RoboDK station: M301_01 v3.rdk

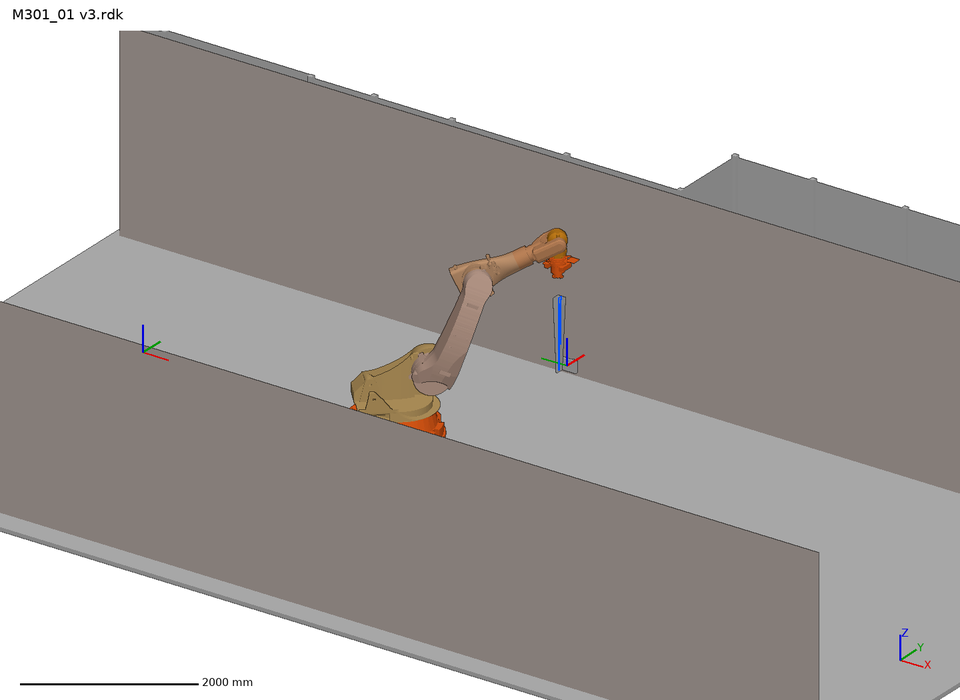
[picture v0: the station drawn from its stored meshes, robots at their saved joint values, targets as dots, program paths as lines]
Station CTTLab. Poses are relative to the parent item; angles as X-Y-Z fixed-axis rotations.
  - object PLANCHER at (0, 0, 0) mm, size 14365 x 8134 x 50 mm, geometry from PLANCHER.STL
  - object BARRIERE_POTEAU at (0, 0, 0) mm, size 13974 x 1274 x 2640 mm, geometry from BARRIERE_POTEAU.STL
  - object BARRIERE_GRILLAGE at (0, 0, 0) mm, size 13811.6 x 1129 x 2475 mm, geometry from BARRIERE_GRILLAGE.STL
  - object BARRIERE_IMMATERIELLE at (0, 0, 0) mm, size 14165 x 6570 x 2640 mm, geometry from BARRIERE_IMMATERIELLE.STL
  - frame World Base at (0, 0, 2.5) mm
    - robot Linear Rail: 1 axes
        modified DH rows (alpha deg, a mm, theta deg, d mm): 0, 0, 0, 0 linear
        base shift (0, 0, 0) mm, rotated rx 0 ry 90 rz 0 deg
        joint limits [0] to [7000]; home [0]; saved at [3500]
      - robot KUKA KR 100 HA: 6 axes
          modified DH rows (alpha deg, a mm, theta deg, d mm): 0, 0, 0, 750; -90, 350, 0, 0; 0, 1250, -90, 0; -90, -45, 0, 1000; 90, 0, 0, 0; -90, 0, 180, 210
          joint limits [-185, -120, -119, -350, -125, -350] to [185, 70, 155, 350, 125, 350]; home [0, -90, 90, 0, 0, 0]; saved at [-41.564, -65.811, 41.041, 0, 114.77, -131.564]
        - tool Tool 1, TCP at (13, 8, 496) mm, size 290.8 x 416.4 x 279.8 mm, geometry from OUTIL.STL
          - object M301_01 at (0, 0, 0) mm, size 101.6 x 101.6 x 914.4 mm, geometry from M301_01.stl
  - frame Camera base at (4846.59, 1350.74, 651.46) mm, rotated rx 0 ry 0 rz 90 deg
    - object Camera at (0, 0, 0) mm, rotated rx 90 ry 0 rz 90 deg, size 220 x 170 x 50 mm, geometry from Camera.stl
    - target Approach target (Cartesian target) at (-112.7, 0, 313.4) mm, rotated rx -180 ry 0 rz -90 deg; joints [-43.056, -66.41, 76.951, 0, 79.459, 136.944, 3500] of KUKA KR 100 HA
    - target Target 0 (Cartesian target) at (-112.7, 0, 881.94) mm, rotated rx -180 ry 0 rz -90 deg; joints [-43.056, -64.348, 40.687, 0, 113.661, 136.944, 3500] of KUKA KR 100 HA
    - target Target 1 (Cartesian target) at (-124.95, 0, 850.56) mm, rotated rx -180 ry 0 rz -90 deg; joints [-42.537, -65.949, 45.083, -0.648, 110.311, 137.463, 3500] of KUKA KR 100 HA
    - target Target 2 (Cartesian target) at (-139.47, 0, 817.45) mm, rotated rx -177.14 ry 0 rz -90 deg; joints [-41.911, -67.558, 49.528, -1.405, 106.807, 137.413, 3500] of KUKA KR 100 HA
    - target Target 3 (Cartesian target) at (-154.54, 0, 817.31) mm, rotated rx -177.14 ry 0 rz -90 deg; joints [-41.235, -68.595, 51.082, -2.235, 105.614, 138.127, 3500] of KUKA KR 100 HA
    - target Target 4 (Cartesian target) at (-154.54, 0, 785.81) mm, rotated rx -177.14 ry 0 rz -90 deg; joints [-41.235, -69.02, 53.562, -2.214, 103.561, 138.21, 3500] of KUKA KR 100 HA
    - target Target 5 (Cartesian target) at (-154.54, 0, 785.81) mm, rotated rx -177.14 ry 0 rz -90 deg; joints [-41.235, -69.02, 53.562, -2.214, 103.561, 138.21, 3500] of KUKA KR 100 HA
    - target Target 6 (Cartesian target) at (-154.54, 0, 754.31) mm, rotated rx -177.14 ry 0 rz -90 deg; joints [-41.235, -69.373, 55.917, -2.197, 101.559, 138.289, 3500] of KUKA KR 100 HA
    - target Target 7 (Cartesian target) at (-154.54, 0, 754.31) mm, rotated rx -177.14 ry 0 rz -90 deg; joints [-41.235, -69.373, 55.917, -2.197, 101.559, 138.289, 3500] of KUKA KR 100 HA
    - target Target 8 (Cartesian target) at (-154.54, 0, 722.81) mm, rotated rx -177.14 ry 0 rz -90 deg; joints [-41.235, -69.661, 58.163, -2.183, 99.603, 138.365, 3500] of KUKA KR 100 HA
    - target Target 9 (Cartesian target) at (-154.54, 0, 722.81) mm, rotated rx -177.14 ry 0 rz -90 deg; joints [-41.235, -69.661, 58.163, -2.183, 99.603, 138.365, 3500] of KUKA KR 100 HA
    - target Target 10 (Cartesian target) at (-154.54, 0, 691.3) mm, rotated rx -177.14 ry 0 rz -90 deg; joints [-41.235, -69.887, 60.31, -2.172, 97.685, 138.439, 3500] of KUKA KR 100 HA
    - target Target 11 (Cartesian target) at (-154.54, 0, 691.3) mm, rotated rx -177.14 ry 0 rz -90 deg; joints [-41.235, -69.887, 60.31, -2.172, 97.685, 138.439, 3500] of KUKA KR 100 HA
    - target Target 12 (Cartesian target) at (-154.54, 0, 659.8) mm, rotated rx -177.14 ry 0 rz -90 deg; joints [-41.235, -70.057, 62.366, -2.163, 95.8, 138.51, 3500] of KUKA KR 100 HA
    - target Target 13 (Cartesian target) at (-154.54, 0, 659.8) mm, rotated rx -177.14 ry 0 rz -90 deg; joints [-41.235, -70.057, 62.366, -2.163, 95.8, 138.51, 3500] of KUKA KR 100 HA
    - target Target 14 (Cartesian target) at (-154.54, 0, 628.3) mm, rotated rx -177.14 ry 0 rz -90 deg; joints [-41.235, -70.173, 64.338, -2.157, 93.944, 138.581, 3500] of KUKA KR 100 HA
    - target Target 15 (Cartesian target) at (-154.54, 0, 628.3) mm, rotated rx -177.14 ry 0 rz -90 deg; joints [-41.235, -70.173, 64.338, -2.157, 93.944, 138.581, 3500] of KUKA KR 100 HA
    - target Target 16 (Cartesian target) at (-154.54, 0, 596.8) mm, rotated rx -177.14 ry 0 rz -90 deg; joints [-41.235, -70.236, 66.234, -2.154, 92.114, 138.65, 3500] of KUKA KR 100 HA
    - target Target 17 (Cartesian target) at (-154.54, 0, 596.8) mm, rotated rx -177.14 ry 0 rz -90 deg; joints [-41.235, -70.236, 66.234, -2.154, 92.114, 138.65, 3500] of KUKA KR 100 HA
    - target Target 18 (Cartesian target) at (-154.54, 0, 565.3) mm, rotated rx -177.14 ry 0 rz -90 deg; joints [-41.235, -70.25, 68.057, -2.152, 90.306, 138.718, 3500] of KUKA KR 100 HA
    - target Target 19 (Cartesian target) at (-154.54, 0, 565.3) mm, rotated rx -177.14 ry 0 rz -90 deg; joints [-41.235, -70.25, 68.057, -2.152, 90.306, 138.718, 3500] of KUKA KR 100 HA
    - target Target 20 (Cartesian target) at (-154.54, 0, 533.8) mm, rotated rx -177.14 ry 0 rz -90 deg; joints [-41.235, -70.216, 69.812, -2.153, 88.518, 138.785, 3500] of KUKA KR 100 HA
    - target Target 21 (Cartesian target) at (-154.54, 0, 533.8) mm, rotated rx -177.14 ry 0 rz -90 deg; joints [-41.235, -70.216, 69.812, -2.153, 88.518, 138.785, 3500] of KUKA KR 100 HA
    - target Target 22 (Cartesian target) at (-154.54, 0, 502.3) mm, rotated rx -177.14 ry 0 rz -90 deg; joints [-41.235, -70.136, 71.503, -2.156, 86.747, 138.851, 3500] of KUKA KR 100 HA
    - target Target 23 (Cartesian target) at (-154.54, 0, 502.3) mm, rotated rx -177.14 ry 0 rz -90 deg; joints [-41.235, -70.136, 71.503, -2.156, 86.747, 138.851, 3500] of KUKA KR 100 HA
    - target Target 24 (Cartesian target) at (-154.54, 0, 470.79) mm, rotated rx -177.14 ry 0 rz -90 deg; joints [-41.235, -70.01, 73.133, -2.16, 84.993, 138.918, 3500] of KUKA KR 100 HA
    - target Target 25 (Cartesian target) at (-154.54, 0, 470.79) mm, rotated rx -177.14 ry 0 rz -90 deg; joints [-41.235, -70.01, 73.133, -2.16, 84.993, 138.918, 3500] of KUKA KR 100 HA
    - target Target 26 (Cartesian target) at (-154.54, 0, 439.29) mm, rotated rx -177.14 ry 0 rz -90 deg; joints [-41.235, -69.84, 74.705, -2.167, 83.252, 138.984, 3500] of KUKA KR 100 HA
    - target Target 27 (Cartesian target) at (-154.54, 0, 439.29) mm, rotated rx -177.14 ry 0 rz -90 deg; joints [-41.235, -69.84, 74.705, -2.167, 83.252, 138.984, 3500] of KUKA KR 100 HA
    - target Target 28 (Cartesian target) at (-154.54, 0, 407.79) mm, rotated rx -177.14 ry 0 rz -90 deg; joints [-41.235, -69.627, 76.221, -2.176, 81.524, 139.05, 3500] of KUKA KR 100 HA
    - target Target 29 (Cartesian target) at (-154.54, 0, 407.79) mm, rotated rx -177.14 ry 0 rz -90 deg; joints [-41.235, -69.627, 76.221, -2.176, 81.524, 139.05, 3500] of KUKA KR 100 HA
    - target Target 30 (Cartesian target) at (-154.54, 0, 376.29) mm, rotated rx -177.14 ry 0 rz -90 deg; joints [-41.235, -69.371, 77.683, -2.187, 79.808, 139.116, 3500] of KUKA KR 100 HA
    - target Target 31 (Cartesian target) at (-154.54, 0, 376.29) mm, rotated rx -177.14 ry 0 rz -90 deg; joints [-41.235, -69.371, 77.683, -2.187, 79.808, 139.116, 3500] of KUKA KR 100 HA
    - target Target 32 (Cartesian target) at (-154.54, 0, 344.79) mm, rotated rx -177.14 ry 0 rz -90 deg; joints [-41.235, -69.074, 79.092, -2.199, 78.102, 139.183, 3500] of KUKA KR 100 HA
    - target Target 33 (Cartesian target) at (-154.54, 0, 344.79) mm, rotated rx -177.14 ry 0 rz -90 deg; joints [-41.235, -69.074, 79.092, -2.199, 78.102, 139.183, 3500] of KUKA KR 100 HA
    - target Target 34 (Cartesian target) at (-154.54, 0, 313.29) mm, rotated rx -177.14 ry 0 rz -90 deg; joints [-41.235, -68.735, 80.451, -2.214, 76.406, 139.25, 3500] of KUKA KR 100 HA
    - target Target 35 (Cartesian target) at (-154.54, 0, 313.29) mm, rotated rx -177.14 ry 0 rz -90 deg; joints [-41.235, -68.735, 80.451, -2.214, 76.406, 139.25, 3500] of KUKA KR 100 HA
    - target Target 36 (Cartesian target) at (-154.54, 0, 281.79) mm, rotated rx -177.14 ry 0 rz -90 deg; joints [-41.235, -68.356, 81.76, -2.231, 74.719, 139.317, 3500] of KUKA KR 100 HA
    - target Target 37 (Cartesian target) at (-154.54, 0, 281.79) mm, rotated rx -177.14 ry 0 rz -90 deg; joints [-41.235, -68.356, 81.76, -2.231, 74.719, 139.317, 3500] of KUKA KR 100 HA
    - target Target 38 (Cartesian target) at (-154.54, 0, 250.29) mm, rotated rx -177.14 ry 0 rz -90 deg; joints [-41.235, -67.936, 83.021, -2.25, 73.04, 139.386, 3500] of KUKA KR 100 HA
    - target Target 39 (Cartesian target) at (-154.54, 0, 218.78) mm, rotated rx -177.14 ry 0 rz -90 deg; joints [-41.235, -67.477, 84.234, -2.271, 71.37, 139.455, 3500] of KUKA KR 100 HA
    - target Target 40 (Cartesian target) at (-154.54, 0, 218.78) mm, rotated rx -177.14 ry 0 rz -90 deg; joints [-41.235, -67.477, 84.234, -2.271, 71.37, 139.455, 3500] of KUKA KR 100 HA
    - target Target 41 (Cartesian target) at (-154.54, 0, 187.28) mm, rotated rx -177.14 ry 0 rz -90 deg; joints [-41.235, -66.979, 85.4, -2.295, 69.707, 139.525, 3500] of KUKA KR 100 HA
    - target Target 42 (Cartesian target) at (-154.54, 0, 187.28) mm, rotated rx -177.14 ry 0 rz -90 deg; joints [-41.235, -66.979, 85.4, -2.295, 69.707, 139.525, 3500] of KUKA KR 100 HA
    - target Target 43 (Cartesian target) at (-154.54, 0, 155.78) mm, rotated rx -177.14 ry 0 rz -90 deg; joints [-41.235, -66.442, 86.519, -2.32, 68.051, 139.597, 3500] of KUKA KR 100 HA
    - target Target 44 (Cartesian target) at (-154.54, 0, 155.78) mm, rotated rx -177.14 ry 0 rz -90 deg; joints [-41.235, -66.442, 86.519, -2.32, 68.051, 139.597, 3500] of KUKA KR 100 HA
    - target Target 45 (Cartesian target) at (-154.54, 0, 124.28) mm, rotated rx -177.14 ry 0 rz -90 deg; joints [-41.235, -65.867, 87.593, -2.349, 66.403, 139.67, 3500] of KUKA KR 100 HA
    - target Target 46 (Cartesian target) at (-154.54, 0, 124.28) mm, rotated rx -177.14 ry 0 rz -90 deg; joints [-41.235, -65.867, 87.593, -2.349, 66.403, 139.67, 3500] of KUKA KR 100 HA
    - target Target 47 (Cartesian target) at (-154.54, 0, 92.78) mm, rotated rx -177.14 ry 0 rz -90 deg; joints [-41.235, -65.254, 88.622, -2.379, 64.763, 139.744, 3500] of KUKA KR 100 HA
    - target Target 48 (Cartesian target) at (-152.66, 0, 92.8) mm, rotated rx -177.14 ry 0 rz -90 deg; joints [-41.626, -64.816, 87.917, -1.397, 65.788, 139.307, 3500] of KUKA KR 100 HA
    - target Target 49 (Cartesian target) at (-151.82, 0, 63.93) mm, rotated rx -180 ry 0 rz -90 deg; joints [-41.878, -63.949, 88.344, -0.751, 64.989, 138.122, 3500] of KUKA KR 100 HA
    - target Target 50 (Cartesian target) at (-150.8, 0, 32.46) mm, rotated rx -180 ry 0 rz -90 deg; joints [-42.17, -62.942, 88.744, 0, 64.199, 137.83, 3500] of KUKA KR 100 HA
    - target Target 51 (Cartesian target) at (-150.8, 0, 1) mm, rotated rx -180 ry 0 rz -90 deg; joints [-42.17, -62.239, 89.64, 0, 62.599, 137.83, 3500] of KUKA KR 100 HA
    - target Target 52 (Cartesian target) at (-150.8, 0, 1) mm, rotated rx -180 ry 0 rz 180 deg; joints [-41.842, -61.484, 88.373, 0, 63.111, 48.158, 3500] of KUKA KR 100 HA
    - target Target 53 (Cartesian target) at (-150.8, 0, 32.46) mm, rotated rx -180 ry 0 rz 180 deg; joints [-41.842, -62.176, 87.478, 0, 64.699, 48.158, 3500] of KUKA KR 100 HA
    - target Target 54 (Cartesian target) at (-150.8, 0, 63.92) mm, rotated rx -180 ry 0 rz 180 deg; joints [-41.842, -62.833, 86.537, 0, 66.296, 48.158, 3500] of KUKA KR 100 HA
    - target Target 55 (Cartesian target) at (-150.8, 0, 95.39) mm, rotated rx -180 ry 0 rz 180 deg; joints [-41.842, -63.453, 85.55, 0, 67.903, 48.158, 3500] of KUKA KR 100 HA
    - target Target 56 (Cartesian target) at (-150.8, 0, 126.85) mm, rotated rx -180 ry 0 rz 180 deg; joints [-41.842, -64.037, 84.517, 0, 69.52, 48.158, 3500] of KUKA KR 100 HA
    - target Target 57 (Cartesian target) at (-150.8, 0, 158.31) mm, rotated rx -180 ry 0 rz 180 deg; joints [-41.842, -64.584, 83.438, 0, 71.146, 48.158, 3500] of KUKA KR 100 HA
    - target Target 58 (Cartesian target) at (-150.8, 0, 189.77) mm, rotated rx -180 ry 0 rz 180 deg; joints [-41.842, -65.094, 82.313, 0, 72.781, 48.158, 3500] of KUKA KR 100 HA
    - target Target 59 (Cartesian target) at (-150.8, 0, 221.23) mm, rotated rx -180 ry 0 rz 180 deg; joints [-41.842, -65.565, 81.139, 0, 74.426, 48.158, 3500] of KUKA KR 100 HA
    - target Target 60 (Cartesian target) at (-150.8, 0, 252.7) mm, rotated rx -180 ry 0 rz 180 deg; joints [-41.842, -65.997, 79.917, 0, 76.08, 48.158, 3500] of KUKA KR 100 HA
    - target Target 61 (Cartesian target) at (-150.8, 0, 284.16) mm, rotated rx -180 ry 0 rz 180 deg; joints [-41.842, -66.391, 78.646, 0, 77.744, 48.158, 3500] of KUKA KR 100 HA
    - target Target 62 (Cartesian target) at (-150.8, 0, 315.62) mm, rotated rx -180 ry 0 rz 180 deg; joints [-41.842, -66.744, 77.325, 0, 79.419, 48.158, 3500] of KUKA KR 100 HA
    - target Target 63 (Cartesian target) at (-150.8, 0, 347.08) mm, rotated rx -180 ry 0 rz 180 deg; joints [-41.842, -67.057, 75.952, 0, 81.106, 48.158, 3500] of KUKA KR 100 HA
    - target Target 64 (Cartesian target) at (-150.8, 0, 378.54) mm, rotated rx -180 ry 0 rz 180 deg; joints [-41.842, -67.329, 74.525, 0, 82.804, 48.158, 3500] of KUKA KR 100 HA
    - target Target 65 (Cartesian target) at (-150.8, 0, 410.01) mm, rotated rx -180 ry 0 rz 180 deg; joints [-41.842, -67.559, 73.044, 0, 84.515, 48.158, 3500] of KUKA KR 100 HA
    - target Target 66 (Cartesian target) at (-150.8, 0, 441.47) mm, rotated rx -180 ry 0 rz 180 deg; joints [-41.842, -67.746, 71.505, 0, 86.241, 48.158, 3500] of KUKA KR 100 HA
    - target Target 67 (Cartesian target) at (-150.8, 0, 472.93) mm, rotated rx -180 ry 0 rz 180 deg; joints [-41.842, -67.89, 69.908, 0, 87.982, 48.158, 3500] of KUKA KR 100 HA
    - target Target 68 (Cartesian target) at (-150.8, 0, 504.39) mm, rotated rx -180 ry 0 rz 180 deg; joints [-41.842, -67.988, 68.248, 0, 89.741, 48.158, 3500] of KUKA KR 100 HA
    - target Target 69 (Cartesian target) at (-150.8, 0, 535.86) mm, rotated rx -180 ry 0 rz 180 deg; joints [-41.842, -68.04, 66.522, 0, 91.518, 48.158, 3500] of KUKA KR 100 HA
    - target Target 70 (Cartesian target) at (-150.8, 0, 567.32) mm, rotated rx -180 ry 0 rz 180 deg; joints [-41.842, -68.045, 64.728, 0, 93.317, 48.158, 3500] of KUKA KR 100 HA
    - target Target 71 (Cartesian target) at (-150.8, 0, 598.78) mm, rotated rx -180 ry 0 rz 180 deg; joints [-41.842, -67.999, 62.86, 0, 95.14, 48.158, 3500] of KUKA KR 100 HA
    - target Target 72 (Cartesian target) at (-150.8, 0, 630.24) mm, rotated rx -180 ry 0 rz 180 deg; joints [-41.842, -67.902, 60.912, 0, 96.99, 48.158, 3500] of KUKA KR 100 HA
    - target Target 73 (Cartesian target) at (-150.8, 0, 661.7) mm, rotated rx -180 ry 0 rz 180 deg; joints [-41.842, -67.75, 58.88, 0, 98.87, 48.158, 3500] of KUKA KR 100 HA
    - target Target 74 (Cartesian target) at (-150.8, 0, 693.17) mm, rotated rx -180 ry 0 rz 180 deg; joints [-41.842, -67.541, 56.755, 0, 100.786, 48.158, 3500] of KUKA KR 100 HA
    - target Target 75 (Cartesian target) at (-150.8, 0, 724.63) mm, rotated rx -180 ry 0 rz 180 deg; joints [-41.842, -67.27, 54.528, 0, 102.742, 48.158, 3500] of KUKA KR 100 HA
    - target Target 76 (Cartesian target) at (-150.8, 0, 756.09) mm, rotated rx -180 ry 0 rz 180 deg; joints [-41.842, -66.933, 52.188, 0, 104.745, 48.158, 3500] of KUKA KR 100 HA
    - target Target 77 (Cartesian target) at (-150.8, 0, 787.55) mm, rotated rx -180 ry 0 rz 180 deg; joints [-41.842, -66.524, 49.722, 0, 106.802, 48.158, 3500] of KUKA KR 100 HA
    - target Target 78 (Cartesian target) at (-150.8, 0, 819.01) mm, rotated rx -180 ry 0 rz 180 deg; joints [-41.842, -66.034, 47.111, 0, 108.924, 48.158, 3500] of KUKA KR 100 HA
    - target Target 79 (Cartesian target) at (-150.8, 0, 850.48) mm, rotated rx -180 ry 0 rz 180 deg; joints [-41.842, -65.455, 44.332, 0, 111.123, 48.158, 3500] of KUKA KR 100 HA
    - target Target 80 (Cartesian target) at (-150.8, 0, 881.94) mm, rotated rx -180 ry 0 rz 180 deg; joints [-41.842, -64.773, 41.356, 0, 113.417, 48.158, 3500] of KUKA KR 100 HA
    - target Target 81 (Cartesian target) at (-150.8, 0, 913.4) mm, rotated rx -180 ry 0 rz 180 deg; joints [-41.842, -63.969, 38.141, 0, 115.828, 48.158, 3500] of KUKA KR 100 HA
    - target Target 82 (Cartesian target) at (-112.7, 0, 913.4) mm, rotated rx -180 ry 0 rz 90 deg; joints [-42.136, -62.977, 36.545, 0, 116.432, -42.136, 3500] of KUKA KR 100 HA
    - target Target 83 (Cartesian target) at (-112.7, 0, 881.94) mm, rotated rx -180 ry 0 rz 90 deg; joints [-42.136, -63.826, 39.86, 0, 113.966, -42.136, 3500] of KUKA KR 100 HA
    - target Target 84 (Cartesian target) at (-124.95, 0, 850.56) mm, rotated rx -180 ry 0 rz 90 deg; joints [-41.612, -65.441, 44.3, -0.659, 110.596, -41.612, 3500] of KUKA KR 100 HA
    - target Target 85 (Cartesian target) at (-139.47, 0, 817.45) mm, rotated rx 177.14 ry 0 rz 90 deg; joints [-40.979, -67.07, 48.843, -1.427, 107.026, -41.674, 3500] of KUKA KR 100 HA
    - target Target 86 (Cartesian target) at (-154.54, 0, 817.31) mm, rotated rx 177.14 ry 0 rz 90 deg; joints [-40.298, -68.096, 50.392, -2.269, 105.84, -40.953, 3500] of KUKA KR 100 HA
    - target Target 87 (Cartesian target) at (-154.54, 0, 785.81) mm, rotated rx 177.14 ry 0 rz 90 deg; joints [-40.298, -68.53, 52.891, -2.247, 103.776, -40.869, 3500] of KUKA KR 100 HA
    - target Target 88 (Cartesian target) at (-154.54, 0, 785.81) mm, rotated rx 177.14 ry 0 rz 90 deg; joints [-40.298, -68.53, 52.891, -2.247, 103.776, -40.869, 3500] of KUKA KR 100 HA
    - target Target 89 (Cartesian target) at (-154.54, 0, 754.31) mm, rotated rx 177.14 ry 0 rz 90 deg; joints [-40.298, -68.891, 55.263, -2.23, 101.766, -40.788, 3500] of KUKA KR 100 HA
    - target Target 90 (Cartesian target) at (-154.54, 0, 754.31) mm, rotated rx 177.14 ry 0 rz 90 deg; joints [-40.298, -68.891, 55.263, -2.23, 101.766, -40.788, 3500] of KUKA KR 100 HA
    - target Target 91 (Cartesian target) at (-154.54, 0, 722.81) mm, rotated rx 177.14 ry 0 rz 90 deg; joints [-40.298, -69.185, 57.523, -2.215, 99.803, -40.711, 3500] of KUKA KR 100 HA
    - target Target 92 (Cartesian target) at (-154.54, 0, 722.81) mm, rotated rx 177.14 ry 0 rz 90 deg; joints [-40.298, -69.185, 57.523, -2.215, 99.803, -40.711, 3500] of KUKA KR 100 HA
    - target Target 93 (Cartesian target) at (-154.54, 0, 691.3) mm, rotated rx 177.14 ry 0 rz 90 deg; joints [-40.298, -69.418, 59.681, -2.204, 97.879, -40.636, 3500] of KUKA KR 100 HA
    - target Target 94 (Cartesian target) at (-154.54, 0, 691.3) mm, rotated rx 177.14 ry 0 rz 90 deg; joints [-40.298, -69.418, 59.681, -2.204, 97.879, -40.636, 3500] of KUKA KR 100 HA
    - target Target 95 (Cartesian target) at (-154.54, 0, 659.8) mm, rotated rx 177.14 ry 0 rz 90 deg; joints [-40.298, -69.593, 61.747, -2.195, 95.99, -40.563, 3500] of KUKA KR 100 HA
    - target Target 96 (Cartesian target) at (-154.54, 0, 659.8) mm, rotated rx 177.14 ry 0 rz 90 deg; joints [-40.298, -69.593, 61.747, -2.195, 95.99, -40.563, 3500] of KUKA KR 100 HA
    - target Target 97 (Cartesian target) at (-154.54, 0, 628.3) mm, rotated rx 177.14 ry 0 rz 90 deg; joints [-40.298, -69.713, 63.728, -2.188, 94.13, -40.491, 3500] of KUKA KR 100 HA
    - target Target 98 (Cartesian target) at (-154.54, 0, 628.3) mm, rotated rx 177.14 ry 0 rz 90 deg; joints [-40.298, -69.713, 63.728, -2.188, 94.13, -40.491, 3500] of KUKA KR 100 HA
    - target Target 99 (Cartesian target) at (-154.54, 0, 596.8) mm, rotated rx 177.14 ry 0 rz 90 deg; joints [-40.298, -69.781, 65.63, -2.184, 92.297, -40.421, 3500] of KUKA KR 100 HA
    - target Target 100 (Cartesian target) at (-154.54, 0, 596.8) mm, rotated rx 177.14 ry 0 rz 90 deg; joints [-40.298, -69.781, 65.63, -2.184, 92.297, -40.421, 3500] of KUKA KR 100 HA
    - target Target 101 (Cartesian target) at (-154.54, 0, 565.3) mm, rotated rx 177.14 ry 0 rz 90 deg; joints [-40.298, -69.8, 67.459, -2.183, 90.488, -40.352, 3500] of KUKA KR 100 HA
    - target Target 102 (Cartesian target) at (-154.54, 0, 565.3) mm, rotated rx 177.14 ry 0 rz 90 deg; joints [-40.298, -69.8, 67.459, -2.183, 90.488, -40.352, 3500] of KUKA KR 100 HA
    - target Target 103 (Cartesian target) at (-154.54, 0, 533.8) mm, rotated rx 177.14 ry 0 rz 90 deg; joints [-40.298, -69.769, 69.22, -2.183, 88.698, -40.284, 3500] of KUKA KR 100 HA
    - target Target 104 (Cartesian target) at (-154.54, 0, 533.8) mm, rotated rx 177.14 ry 0 rz 90 deg; joints [-40.298, -69.769, 69.22, -2.183, 88.698, -40.284, 3500] of KUKA KR 100 HA
    - target Target 105 (Cartesian target) at (-154.54, 0, 502.3) mm, rotated rx 177.14 ry 0 rz 90 deg; joints [-40.298, -69.692, 70.915, -2.186, 86.928, -40.216, 3500] of KUKA KR 100 HA
    - target Target 106 (Cartesian target) at (-154.54, 0, 502.3) mm, rotated rx 177.14 ry 0 rz 90 deg; joints [-40.298, -69.692, 70.915, -2.186, 86.928, -40.216, 3500] of KUKA KR 100 HA
    - target Target 107 (Cartesian target) at (-154.54, 0, 470.79) mm, rotated rx 177.14 ry 0 rz 90 deg; joints [-40.298, -69.57, 72.548, -2.191, 85.173, -40.149, 3500] of KUKA KR 100 HA
    - target Target 108 (Cartesian target) at (-154.54, 0, 470.79) mm, rotated rx 177.14 ry 0 rz 90 deg; joints [-40.298, -69.57, 72.548, -2.191, 85.173, -40.149, 3500] of KUKA KR 100 HA
    - target Target 109 (Cartesian target) at (-154.54, 0, 439.29) mm, rotated rx 177.14 ry 0 rz 90 deg; joints [-40.298, -69.404, 74.123, -2.197, 83.433, -40.082, 3500] of KUKA KR 100 HA
    - target Target 110 (Cartesian target) at (-154.54, 0, 439.29) mm, rotated rx 177.14 ry 0 rz 90 deg; joints [-40.298, -69.404, 74.123, -2.197, 83.433, -40.082, 3500] of KUKA KR 100 HA
    - target Target 111 (Cartesian target) at (-154.54, 0, 407.79) mm, rotated rx 177.14 ry 0 rz 90 deg; joints [-40.298, -69.194, 75.641, -2.206, 81.706, -40.015, 3500] of KUKA KR 100 HA
    - target Target 112 (Cartesian target) at (-154.54, 0, 407.79) mm, rotated rx 177.14 ry 0 rz 90 deg; joints [-40.298, -69.194, 75.641, -2.206, 81.706, -40.015, 3500] of KUKA KR 100 HA
    - target Target 113 (Cartesian target) at (-154.54, 0, 376.29) mm, rotated rx 177.14 ry 0 rz 90 deg; joints [-40.298, -68.941, 77.104, -2.216, 79.992, -39.948, 3500] of KUKA KR 100 HA
    - target Target 114 (Cartesian target) at (-154.54, 0, 376.29) mm, rotated rx 177.14 ry 0 rz 90 deg; joints [-40.298, -68.941, 77.104, -2.216, 79.992, -39.948, 3500] of KUKA KR 100 HA
    - target Target 115 (Cartesian target) at (-154.54, 0, 344.79) mm, rotated rx 177.14 ry 0 rz 90 deg; joints [-40.298, -68.647, 78.515, -2.229, 78.288, -39.881, 3500] of KUKA KR 100 HA
    - target Target 116 (Cartesian target) at (-154.54, 0, 344.79) mm, rotated rx 177.14 ry 0 rz 90 deg; joints [-40.298, -68.647, 78.515, -2.229, 78.288, -39.881, 3500] of KUKA KR 100 HA
    - target Target 117 (Cartesian target) at (-154.54, 0, 313.29) mm, rotated rx 177.14 ry 0 rz 90 deg; joints [-40.298, -68.311, 79.875, -2.244, 76.594, -39.813, 3500] of KUKA KR 100 HA
    - target Target 118 (Cartesian target) at (-154.54, 0, 313.29) mm, rotated rx 177.14 ry 0 rz 90 deg; joints [-40.298, -68.311, 79.875, -2.244, 76.594, -39.813, 3500] of KUKA KR 100 HA
    - target Target 119 (Cartesian target) at (-154.54, 0, 281.79) mm, rotated rx 177.14 ry 0 rz 90 deg; joints [-40.298, -67.935, 81.184, -2.261, 74.91, -39.745, 3500] of KUKA KR 100 HA
    - target Target 120 (Cartesian target) at (-154.54, 0, 281.79) mm, rotated rx 177.14 ry 0 rz 90 deg; joints [-40.298, -67.935, 81.184, -2.261, 74.91, -39.745, 3500] of KUKA KR 100 HA
    - target Target 121 (Cartesian target) at (-154.54, 0, 250.29) mm, rotated rx 177.14 ry 0 rz 90 deg; joints [-40.298, -67.519, 82.445, -2.28, 73.235, -39.676, 3500] of KUKA KR 100 HA
    - target Target 122 (Cartesian target) at (-154.54, 0, 218.78) mm, rotated rx 177.14 ry 0 rz 90 deg; joints [-40.298, -67.064, 83.657, -2.301, 71.568, -39.606, 3500] of KUKA KR 100 HA
    - target Target 123 (Cartesian target) at (-154.54, 0, 218.78) mm, rotated rx 177.14 ry 0 rz 90 deg; joints [-40.298, -67.064, 83.657, -2.301, 71.568, -39.606, 3500] of KUKA KR 100 HA
    - target Target 124 (Cartesian target) at (-154.54, 0, 187.28) mm, rotated rx 177.14 ry 0 rz 90 deg; joints [-40.298, -66.569, 84.823, -2.324, 69.909, -39.535, 3500] of KUKA KR 100 HA
    - target Target 125 (Cartesian target) at (-154.54, 0, 187.28) mm, rotated rx 177.14 ry 0 rz 90 deg; joints [-40.298, -66.569, 84.823, -2.324, 69.909, -39.535, 3500] of KUKA KR 100 HA
    - target Target 126 (Cartesian target) at (-154.54, 0, 155.78) mm, rotated rx 177.14 ry 0 rz 90 deg; joints [-40.298, -66.036, 85.942, -2.35, 68.259, -39.463, 3500] of KUKA KR 100 HA
    - target Target 127 (Cartesian target) at (-154.54, 0, 155.78) mm, rotated rx 177.14 ry 0 rz 90 deg; joints [-40.298, -66.036, 85.942, -2.35, 68.259, -39.463, 3500] of KUKA KR 100 HA
    - target Target 128 (Cartesian target) at (-154.54, 0, 124.28) mm, rotated rx 177.14 ry 0 rz 90 deg; joints [-40.298, -65.465, 87.015, -2.378, 66.616, -39.389, 3500] of KUKA KR 100 HA
    - target Target 129 (Cartesian target) at (-154.54, 0, 124.28) mm, rotated rx 177.14 ry 0 rz 90 deg; joints [-40.298, -65.465, 87.015, -2.378, 66.616, -39.389, 3500] of KUKA KR 100 HA
    - target Target 130 (Cartesian target) at (-154.54, 0, 92.78) mm, rotated rx 177.14 ry 0 rz 90 deg; joints [-40.298, -64.856, 88.042, -2.409, 64.981, -39.314, 3500] of KUKA KR 100 HA
    - target Target 131 (Cartesian target) at (-152.66, 0, 92.8) mm, rotated rx 177.14 ry 0 rz 90 deg; joints [-40.692, -64.426, 87.347, -1.415, 65.989, -39.754, 3500] of KUKA KR 100 HA
    - target Target 132 (Cartesian target) at (-151.82, 0, 63.93) mm, rotated rx -180 ry 0 rz 90 deg; joints [-40.946, -63.584, 87.754, -0.761, 65.226, -40.946, 3500] of KUKA KR 100 HA
    - target Target 133 (Cartesian target) at (-150.8, 0, 32.46) mm, rotated rx -180 ry 0 rz 90 deg; joints [-41.241, -62.589, 88.16, 0, 64.429, -41.241, 3500] of KUKA KR 100 HA
    - target Target 134 (Cartesian target) at (-150.8, 0, 1) mm, rotated rx -180 ry 0 rz 90 deg; joints [-41.241, -61.89, 89.056, 0, 62.835, -41.241, 3500] of KUKA KR 100 HA
    - target Target 135 (Cartesian target) at (-150.8, 0, 1) mm, rotated rx -180 ry 0 rz 0 deg; joints [-41.564, -62.648, 90.321, 0, 62.327, -131.564, 3500] of KUKA KR 100 HA
    - target Target 136 (Cartesian target) at (-150.8, 0, 32.46) mm, rotated rx -180 ry 0 rz 0 deg; joints [-41.564, -63.357, 89.424, 0, 63.933, -131.564, 3500] of KUKA KR 100 HA
    - target Target 137 (Cartesian target) at (-150.8, 0, 63.92) mm, rotated rx -180 ry 0 rz 0 deg; joints [-41.564, -64.031, 88.483, 0, 65.548, -131.564, 3500] of KUKA KR 100 HA
    - target Target 138 (Cartesian target) at (-150.8, 0, 95.39) mm, rotated rx -180 ry 0 rz 0 deg; joints [-41.564, -64.668, 87.497, 0, 67.171, -131.564, 3500] of KUKA KR 100 HA
    - target Target 139 (Cartesian target) at (-150.8, 0, 126.85) mm, rotated rx -180 ry 0 rz 0 deg; joints [-41.564, -65.268, 86.465, 0, 68.803, -131.564, 3500] of KUKA KR 100 HA
    - target Target 140 (Cartesian target) at (-150.8, 0, 158.31) mm, rotated rx -180 ry 0 rz 0 deg; joints [-41.564, -65.831, 85.388, 0, 70.443, -131.564, 3500] of KUKA KR 100 HA
    - target Target 141 (Cartesian target) at (-150.8, 0, 189.77) mm, rotated rx -180 ry 0 rz 0 deg; joints [-41.564, -66.355, 84.264, 0, 72.091, -131.564, 3500] of KUKA KR 100 HA
    - target Target 142 (Cartesian target) at (-150.8, 0, 221.23) mm, rotated rx -180 ry 0 rz 0 deg; joints [-41.564, -66.841, 83.094, 0, 73.747, -131.564, 3500] of KUKA KR 100 HA
    - target Target 143 (Cartesian target) at (-150.8, 0, 252.7) mm, rotated rx -180 ry 0 rz 0 deg; joints [-41.564, -67.289, 81.877, 0, 75.412, -131.564, 3500] of KUKA KR 100 HA
    - target Target 144 (Cartesian target) at (-150.8, 0, 284.16) mm, rotated rx -180 ry 0 rz 0 deg; joints [-41.564, -67.696, 80.611, 0, 77.085, -131.564, 3500] of KUKA KR 100 HA
    - target Target 145 (Cartesian target) at (-150.8, 0, 315.62) mm, rotated rx -180 ry 0 rz 0 deg; joints [-41.564, -68.064, 79.296, 0, 78.768, -131.564, 3500] of KUKA KR 100 HA
    - target Target 146 (Cartesian target) at (-150.8, 0, 347.08) mm, rotated rx -180 ry 0 rz 0 deg; joints [-41.564, -68.392, 77.931, 0, 80.46, -131.564, 3500] of KUKA KR 100 HA
    - target Target 147 (Cartesian target) at (-150.8, 0, 378.54) mm, rotated rx -180 ry 0 rz 0 deg; joints [-41.564, -68.678, 76.515, 0, 82.163, -131.564, 3500] of KUKA KR 100 HA
    - target Target 148 (Cartesian target) at (-150.8, 0, 410.01) mm, rotated rx -180 ry 0 rz 0 deg; joints [-41.564, -68.922, 75.045, 0, 83.878, -131.564, 3500] of KUKA KR 100 HA
    - target Target 149 (Cartesian target) at (-150.8, 0, 441.47) mm, rotated rx -180 ry 0 rz 0 deg; joints [-41.564, -69.124, 73.52, 0, 85.604, -131.564, 3500] of KUKA KR 100 HA
    - target Target 150 (Cartesian target) at (-150.8, 0, 472.93) mm, rotated rx -180 ry 0 rz 0 deg; joints [-41.564, -69.283, 71.938, 0, 87.345, -131.564, 3500] of KUKA KR 100 HA
    - target Target 151 (Cartesian target) at (-150.8, 0, 504.39) mm, rotated rx -180 ry 0 rz 0 deg; joints [-41.564, -69.397, 70.296, 0, 89.101, -131.564, 3500] of KUKA KR 100 HA
    - target Target 152 (Cartesian target) at (-150.8, 0, 535.86) mm, rotated rx -180 ry 0 rz 0 deg; joints [-41.564, -69.465, 68.592, 0, 90.873, -131.564, 3500] of KUKA KR 100 HA
    - target Target 153 (Cartesian target) at (-150.8, 0, 567.32) mm, rotated rx -180 ry 0 rz 0 deg; joints [-41.564, -69.487, 66.822, 0, 92.665, -131.564, 3500] of KUKA KR 100 HA
    - target Target 154 (Cartesian target) at (-150.8, 0, 598.78) mm, rotated rx -180 ry 0 rz 0 deg; joints [-41.564, -69.46, 64.982, 0, 94.478, -131.564, 3500] of KUKA KR 100 HA
    - target Target 155 (Cartesian target) at (-150.8, 0, 630.24) mm, rotated rx -180 ry 0 rz 0 deg; joints [-41.564, -69.383, 63.068, 0, 96.315, -131.564, 3500] of KUKA KR 100 HA
    - target Target 156 (Cartesian target) at (-150.8, 0, 661.7) mm, rotated rx -180 ry 0 rz 0 deg; joints [-41.564, -69.253, 61.074, 0, 98.179, -131.564, 3500] of KUKA KR 100 HA
    - target Target 157 (Cartesian target) at (-150.8, 0, 693.17) mm, rotated rx -180 ry 0 rz 0 deg; joints [-41.564, -69.067, 58.993, 0, 100.075, -131.564, 3500] of KUKA KR 100 HA
    - target Target 158 (Cartesian target) at (-150.8, 0, 724.63) mm, rotated rx -180 ry 0 rz 0 deg; joints [-41.564, -68.824, 56.817, 0, 102.006, -131.564, 3500] of KUKA KR 100 HA
    - target Target 159 (Cartesian target) at (-150.8, 0, 756.09) mm, rotated rx -180 ry 0 rz 0 deg; joints [-41.564, -68.517, 54.538, 0, 103.979, -131.564, 3500] of KUKA KR 100 HA
    - target Target 160 (Cartesian target) at (-150.8, 0, 787.55) mm, rotated rx -180 ry 0 rz 0 deg; joints [-41.564, -68.143, 52.143, 0, 106, -131.564, 3500] of KUKA KR 100 HA
    - target Target 161 (Cartesian target) at (-150.8, 0, 819.01) mm, rotated rx -180 ry 0 rz 0 deg; joints [-41.564, -67.694, 49.618, 0, 108.077, -131.564, 3500] of KUKA KR 100 HA
    - target Target 162 (Cartesian target) at (-150.8, 0, 850.48) mm, rotated rx -180 ry 0 rz 0 deg; joints [-41.564, -67.164, 46.943, 0, 110.221, -131.564, 3500] of KUKA KR 100 HA
    - target Target 163 (Cartesian target) at (-150.8, 0, 881.94) mm, rotated rx -180 ry 0 rz 0 deg; joints [-41.564, -66.541, 44.095, 0, 112.446, -131.564, 3500] of KUKA KR 100 HA
    - target Target 164 (Cartesian target) at (-150.8, 0, 913.4) mm, rotated rx -180 ry 0 rz 0 deg; joints [-41.564, -65.811, 41.041, 0, 114.77, -131.564, 3500] of KUKA KR 100 HA
  - Python program LoadProgram (listed below)
  - Python program SearchExternalJoints (listed below)
  - program M301_01 Picture Analysis (169 instructions, listed below)
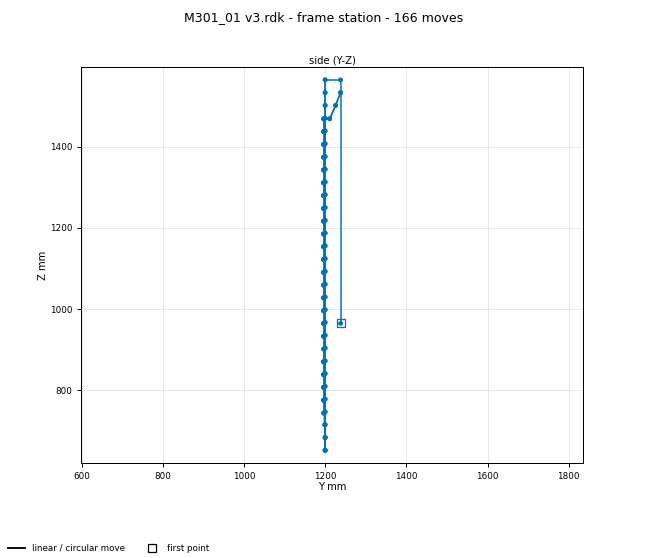
[picture p0: tool path of M301_01 v3.rdk in frame station, 166 of 166 moves have a stored position in this frame; points joined in program order, loops and branches not executed]

--- Python program LoadProgram ---
from robolink import *

RDK = Robolink()

robot = RDK.Item('KUKA KR 100 HA', ITEM_TYPE_ROBOT)
if not robot.Valid():
    raise Exception('No robot selected or available')

world_base = RDK.Item('World Base', ITEM_TYPE_FRAME)
camera_base = RDK.Item('Camera base', ITEM_TYPE_FRAME)
tool = RDK.Item('Tool 1', ITEM_TYPE_TOOL)

RDK.Render(False)


# Specify the reference frame you want to use
program = RDK.AddProgram("{} Picture Analysis".format(name_prog), robot)
program.setPoseFrame(camera_base)
program.setPoseTool(tool)

program.setSpeed(speed, 200, 10000, 800)

target_name = 'Approach target'
pose = Mat(htm[0].tolist())
target = RDK.AddTarget(target_name, camera_base, tool)
target.setAsCartesianTarget()
target.setPose(pose)
program.MoveJ(target)



for i in range(htm.shape[0] - 1):
    target_name = 'Target {}'.format(i)
    pose = Mat(htm[i + 1].tolist())
    target = RDK.AddTarget(target_name, camera_base, tool)
    e1 = 5000
    target.setJoints([0,0,0,0,0,0, e1])
    target.setAsCartesianTarget()
    target.setPose(pose)
    program.MoveL(target)

--- Python program SearchExternalJoints ---
# Type help("robolink") or help("robodk") for more information
# Press F5 to run the script
# Documentation: https://robodk.com/doc/en/RoboDK-API.html
# Reference:     https://robodk.com/doc/en/PythonAPI/index.html
# Note: It is not required to keep a copy of this file, your python script is saved with the station
from robolink import *    # RoboDK API
from robodk import *      # Robot toolbox
RDK = Robolink()

targets = RDK.ItemList(ITEM_TYPE_TARGET)

# Select a program (automatic selection if you have only one program)
program = RDK.ItemUserPick('Select a program to check and update targets', ITEM_TYPE_PROGRAM)

RDK.Render(False)

# List some candidates for e1:
Test_E1 = [500, 1000, 1500, 2000, 2500, 3000, 3500, 4000, 4500]
#test_E1 = range(500, 5000, 500)

for e1 in Test_E1:
    print("Testing program feasibility for E1:" + str(e1))

    # Update all targets to desired e1
    for t in targets:
        # Set the value of the external axis
        # e1 = 5000 # in mm
        t.setJoints([0,0,0,0,0,0, e1])

        # Recalculate the joint position based on the new position of the external axis
        # Robot joints are updated but not external axis
        t.setAsCartesianTarget()
        t.Joints()

        jnts = t.Joints()
        print(t.Name() + "-Joints: " + str(jnts.list()))

    # Test the program and make sure it is 100% feasible
    valid_ins, prog_time, prog_len, valid_ratio, error_msg = program.Update()
    if valid_ratio < 1.0:
        print("  Unable to complete the program")
        print("  " + error_msg)

    else:
        print("  Program feasible!")
        # stop looking
        break

print("Done!")
program.RunProgram()

--- program M301_01 Picture Analysis (robot KUKA KR 100 HA) ---
  Set Ref.: Camera base
  Choisir Outil: Tool 1
  Set speed (50.0 mm/s)
  MoveJ (Approach target)
  MoveL (Target 0)
  MoveL (Target 1)
  MoveL (Target 2)
  MoveL (Target 3)
  MoveL (Target 4)
  MoveL (Target 5)
  MoveL (Target 6)
  MoveL (Target 7)
  MoveL (Target 8)
  MoveL (Target 9)
  MoveL (Target 10)
  MoveL (Target 11)
  MoveL (Target 12)
  MoveL (Target 13)
  MoveL (Target 14)
  MoveL (Target 15)
  MoveL (Target 16)
  MoveL (Target 17)
  MoveL (Target 18)
  MoveL (Target 19)
  MoveL (Target 20)
  MoveL (Target 21)
  MoveL (Target 22)
  MoveL (Target 23)
  MoveL (Target 24)
  MoveL (Target 25)
  MoveL (Target 26)
  MoveL (Target 27)
  MoveL (Target 28)
  MoveL (Target 29)
  MoveL (Target 30)
  MoveL (Target 31)
  MoveL (Target 32)
  MoveL (Target 33)
  MoveL (Target 34)
  MoveL (Target 35)
  MoveL (Target 36)
  MoveL (Target 37)
  MoveL (Target 38)
  MoveL (Target 39)
  MoveL (Target 40)
  MoveL (Target 41)
  MoveL (Target 42)
  MoveL (Target 43)
  MoveL (Target 44)
  MoveL (Target 45)
  MoveL (Target 46)
  MoveL (Target 47)
  MoveL (Target 48)
  MoveL (Target 49)
  MoveL (Target 50)
  MoveL (Target 51)
  MoveL (Target 52)
  MoveL (Target 53)
  MoveL (Target 54)
  MoveL (Target 55)
  MoveL (Target 56)
  MoveL (Target 57)
  MoveL (Target 58)
  MoveL (Target 59)
  MoveL (Target 60)
  MoveL (Target 61)
  MoveL (Target 62)
  MoveL (Target 63)
  MoveL (Target 64)
  MoveL (Target 65)
  MoveL (Target 66)
  MoveL (Target 67)
  MoveL (Target 68)
  MoveL (Target 69)
  MoveL (Target 70)
  MoveL (Target 71)
  MoveL (Target 72)
  MoveL (Target 73)
  MoveL (Target 74)
  MoveL (Target 75)
  MoveL (Target 76)
  MoveL (Target 77)
  MoveL (Target 78)
  MoveL (Target 79)
  MoveL (Target 80)
  MoveL (Target 81)
  MoveL (Target 82)
  MoveL (Target 83)
  MoveL (Target 84)
  MoveL (Target 85)
  MoveL (Target 86)
  MoveL (Target 87)
  MoveL (Target 88)
  MoveL (Target 89)
  MoveL (Target 90)
  MoveL (Target 91)
  MoveL (Target 92)
  MoveL (Target 93)
  MoveL (Target 94)
  MoveL (Target 95)
  MoveL (Target 96)
  MoveL (Target 97)
  MoveL (Target 98)
  MoveL (Target 99)
  MoveL (Target 100)
  MoveL (Target 101)
  MoveL (Target 102)
  MoveL (Target 103)
  MoveL (Target 104)
  MoveL (Target 105)
  MoveL (Target 106)
  MoveL (Target 107)
  MoveL (Target 108)
  MoveL (Target 109)
  MoveL (Target 110)
  MoveL (Target 111)
  MoveL (Target 112)
  MoveL (Target 113)
  MoveL (Target 114)
  MoveL (Target 115)
  MoveL (Target 116)
  MoveL (Target 117)
  MoveL (Target 118)
  MoveL (Target 119)
  MoveL (Target 120)
  MoveL (Target 121)
  MoveL (Target 122)
  MoveL (Target 123)
  MoveL (Target 124)
  MoveL (Target 125)
  MoveL (Target 126)
  MoveL (Target 127)
  MoveL (Target 128)
  MoveL (Target 129)
  MoveL (Target 130)
  MoveL (Target 131)
  MoveL (Target 132)
  MoveL (Target 133)
  MoveL (Target 134)
  MoveL (Target 135)
  MoveL (Target 136)
  MoveL (Target 137)
  MoveL (Target 138)
  MoveL (Target 139)
  MoveL (Target 140)
  MoveL (Target 141)
  MoveL (Target 142)
  MoveL (Target 143)
  MoveL (Target 144)
  MoveL (Target 145)
  MoveL (Target 146)
  MoveL (Target 147)
  MoveL (Target 148)
  MoveL (Target 149)
  MoveL (Target 150)
  MoveL (Target 151)
  MoveL (Target 152)
  MoveL (Target 153)
  MoveL (Target 154)
  MoveL (Target 155)
  MoveL (Target 156)
  MoveL (Target 157)
  MoveL (Target 158)
  MoveL (Target 159)
  MoveL (Target 160)
  MoveL (Target 161)
  MoveL (Target 162)
  MoveL (Target 163)
  MoveL (Target 164)
